// TIA Portal project "2022.06.13_步进电机定位指令2" (V17)

(* hardware
DEVICE "S7-1200 station_1"  S7-1200 Station
   slot 0: "Rack_0"  S7-1200 Rack  Rack  V1.0
   slot 1: "PLC_1"  CPU 1212C DC/DC/DC  6ES7 212-1AE40-0XB0  V4.5
   slot 2: "AI 4x13BIT/AQ 2x14BIT_1"  SM 1234 AI4/AQ2  6ES7 234-4HE30-0XB0  V1.0
*)

// ===== PLC "PLC_1"  CPU 1212C DC/DC/DC =====

VAR_GLOBAL   // PLC tag table "默认变量表"
   "液位测量" AT %IW96 : Word;
   "百分比" AT %MD40 : DWord;
   "模拟量输出通道" AT %MD44 : UDInt;
   "所需频率(1)" AT %MD0 : Real;
   "压力2模拟输入通道" AT %IW100 : Int;
   "液位" AT %MD4 : Real;
   "频率" AT %MD8 : Real;
   "Tag_2" AT %MD12 : Real;
   "模拟量输出" AT %QW96 : Int;
   "设定液位值" AT %MD20 : Real;
   "实际液位值" AT %MD24 : Real;
   "轴_1_脉冲" AT %Q0.0 : Bool;
   "轴_1_方向" AT %Q0.1 : Bool;
   "轴_1_LowHwLimitSwitch" AT %I0.0 : Bool;
   "轴_1_HighHwLimitSwitch" AT %I0.1 : Bool;
   "轴_1_PassiveHomingSwitch" AT %I0.2 : Bool;
   "轴_1_归位开关" AT %I0.3 : Bool;
   "启用轴" AT %M0.0 : Bool;
   "完成位" AT %M0.1 : Bool;
   "Tag_1" AT %M0.2 : Bool;
   "回原点" AT %I1.0 : Bool;
   "Tag_3" AT %M0.4 : Bool;
   "Tag_4" AT %M0.5 : Bool;
   "Tag_5" AT %M0.3 : Bool;
   "触发绝对定位" AT %I1.1 : Bool;
   "Tag_7" AT %M0.6 : Bool;
   "指定位置" AT %MD30 : Real;
   "指定速度" AT %MD34 : Real;
   "Tag_6" AT %M0.7 : Bool;
   "Tag_8" AT %I1.2 : Bool;
   "Tag_9" AT %M1.0 : Bool;
   "触发相对位移指令" AT %I1.3 : Bool;
   "Tag_11" AT %M1.1 : Bool;
   "相对位置" AT %MD28 : Real;
   "速度" AT %MD32 : Real;
   "触发恒速" AT %I0.4 : Bool;
   "Tag_10" AT %M1.2 : Bool;
   "Tag_12" AT %MD36 : Real;
   "Tag_13" AT %I1.5 : Bool;
   "Tag_14" AT %M1.3 : Bool;
   "正点动" AT %I1.6 : Bool;
   "反点动" AT %I1.7 : Bool;
   "System_Byte" AT %MB100 : Byte;
   "FirstScan" AT %M100.0 : Bool;
   "DiagStatusUpdate" AT %M100.1 : Bool;
   "AlwaysTRUE" AT %M100.2 : Bool;
   "AlwaysFALSE" AT %M100.3 : Bool;
   "Tag_15" AT %M10.0 : Bool;
   "Tag_16" AT %M70.0 : Bool;
   "Tag_17" AT %M70.1 : Bool;
   "Tag_18" AT %M70.2 : Bool;
END_VAR

// folder: System blocks/Program resources

DATA_BLOCK "IEC_Timer_0_DB"   // DB13
{ S7_Optimized_Access := 'TRUE' }
AUTHOR : Simatic
FAMILY : IEC
NAME : IEC_TMR
VERSION : 1.0
// stored: InstanceOfName IEC_TIMER
"IEC_TIMER"
BEGIN
END_DATA_BLOCK

// folder: (top level)

DATA_BLOCK "轴_1"   // DB2, Motion_DB
{ S7_Optimized_Access := 'TRUE' }
AUTHOR : SIMATIC
FAMILY : BasicMC
NAME : TO_PosAx
VERSION : 8.0
// stored: InstanceOfName TO_PositioningAxis
"TO_PositioningAxis"
BEGIN
   // Axis.HomingReferencePointSwitch_AddressCU = %I0.3
   // Axis.LengthUnitNormalized.Distance = 1013
   // Axis.PositionLimitsMax_AddressCU = %I0.1
   // Axis.PositionLimitsMin_AddressCU = %I0.0
   // Axis.OnlinePtoModeCU = 16#0000_0002
   // Axis.DirectionOutputEnabledCU = TRUE
   // Axis.SelectedChannel2EnumCU = %Q0.1
   // Axis.SelectedChannel1EnumCU = %Q0.0
   // Pulse.MinDeltaDeltaFrequencyCU = 0.004
   // Pulse.MaxDeltaDeltaFrequencyCU = 1.0E+10
   // Pulse.MinDeltaFrequencyCU = 0.005
   // Pulse.MaxDeltaFrequencyCU = 9.5E+9
   // Pulse.MinFrequencyCU = 1.0
   // Pulse.MaxFrequencyCU = 100000.0
   // Pulse.OutputSourceCU = 16#0000_0000
   // Axis.SelectPTO = 0
END_DATA_BLOCK

ORGANIZATION_BLOCK "Main"   // OB1, LAD, ProgramCycle
TITLE = "Main Program Sweep (Cycle)"
{ S7_Optimized_Access := 'TRUE' }
VERSION : 0.1
   VAR_INPUT
      Initial_Call : Bool;   // Initial call of this OB
      Remanence : Bool;   // =True, if remanent data are available
   END_VAR
   VAR_TEMP   // added for the SCL form of the ladder/FBD networks
      _w1 : Bool;
      _w2 : Bool;
   END_VAR
BEGIN

REGION Network 1
   // 启用轴：m0.0长为0，即常闭点一直触发
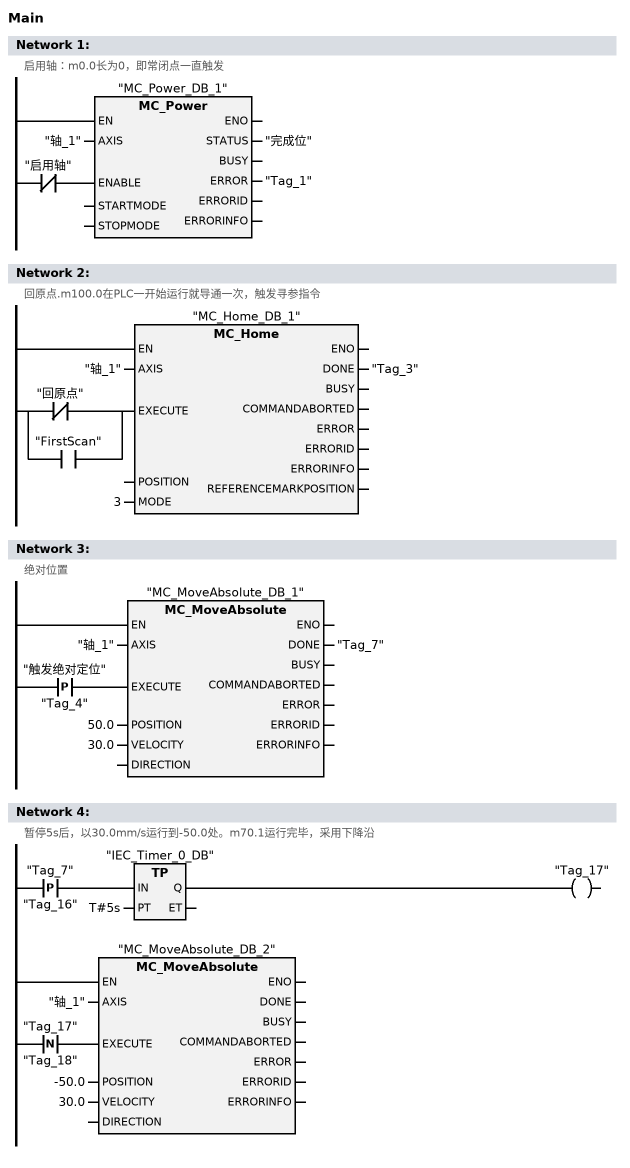
   "MC_Power_DB_1"(Axis := "轴_1", Enable := NOT "启用轴", Status => "完成位", Error => "Tag_1");   // MC_Power
END_REGION

REGION Network 2
   // 回原点.m100.0在PLC一开始运行就导通一次，触发寻参指令
   "MC_Home_DB_1"(Axis := "轴_1", Execute := NOT "回原点" OR "FirstScan", Mode := 3, Done => "Tag_3");   // MC_Home
END_REGION

REGION Network 3
   // 绝对位置
   #_w1 := "触发绝对定位" AND NOT "Tag_4";   // rising edge of "触发绝对定位"
   "Tag_4" := "触发绝对定位";
   "MC_MoveAbsolute_DB_1"(Axis := "轴_1", Execute := #_w1, Position := 50.0, Velocity := 30.0, Done => "Tag_7");   // MC_MoveAbsolute
END_REGION

REGION Network 4
   // 暂停5s后，以30.0mm/s运行到-50.0处。m70.1运行完毕，采用下降沿
   #_w1 := "Tag_7" AND NOT "Tag_16";   // rising edge of "Tag_7"
   "Tag_16" := "Tag_7";
   "IEC_Timer_0_DB".TP(IN := #_w1, PT := T#5s);
   "Tag_17" := "IEC_Timer_0_DB".Q;
   #_w2 := NOT "Tag_17" AND "Tag_18";   // falling edge of "Tag_17"
   "Tag_18" := "Tag_17";
   "MC_MoveAbsolute_DB_2"(Axis := "轴_1", Execute := #_w2, Position := -50.0, Velocity := 30.0);   // MC_MoveAbsolute
END_REGION
END_ORGANIZATION_BLOCK